FUNCTION Convert_DWORD_TO_DT : BOOL
VAR_INPUT
	in : DWORD;
	out : REFERENCE TO DT;
END_VAR
VAR
	converted : DT;
END_VAR

converted := DWORD_TO_DT(in);

IF (DT_TO_DWORD(converted) <> in) THEN
	RETURN;
END_IF

out := converted;
Convert_DWORD_TO_DT := TRUE;

END_FUNCTION

(* stored: Version 1.1.0.1, ProductVersion 3.1.4024.12
   POU Convert_DWORD_TO_DT: Id {e8d77275-2185-4a80-b450-50a395439f2d}, SpecialFunc None *)
